ABB RAPID module: Operations.mod

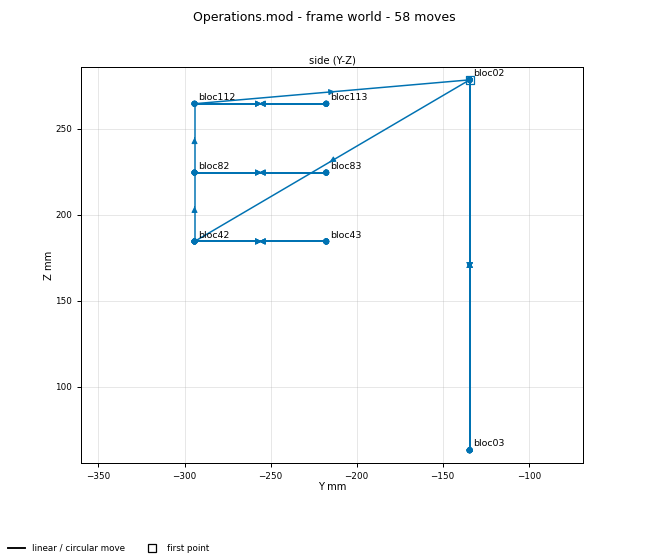
[picture p0: tool path of Operations.mod in frame world, 58 of 59 moves have a stored position in this frame; points joined in program order, loops and branches not executed]
MODULE Operations
 PROC GoHome()
  !
  VAR speeddata HomeSpeed:=[800,100,5000,1000];
  CONST jointtarget PlaceBloc0:=[[-88.65,-2.92,16.23,0,76.69,-88.65],[0,9E9,9E9,9E9,9E9,9E9]];
  MoveAbsJ PlaceBloc0,HomeSpeed,z1,EGP_40_N_N_B;
 ENDPROC
 PROC BuildWall()
  !
  VAR zonedata TransportZone:=[FALSE,5,7.5,7.5,0.75,7.5,0.75];
  VAR speeddata TransportSpeed:=[800,100,5000,1000];
  VAR speeddata PickSpeed:=[60,100,5000,1000];
  CONST robtarget bloc00:=[[-6.5,-340,128.58],[-0.183,-0.683,0.683,0.183],[-1,-1,-2,0],[0,9E9,9E9,9E9,9E9,9E9]];
  CONST robtarget bloc01:=[[-56.5,-340,41.98],[-0.183,-0.683,0.683,0.183],[-1,-1,-2,0],[0,9E9,9E9,9E9,9E9,9E9]];
  CONST robtarget bloc02:=[[211.67,-134.33,278.3],[0.6088,0.7934,0,0],[0,-1,-2,0],[0,9E9,9E9,9E9,9E9,9E9]];
  CONST robtarget bloc03:=[[211.67,-134.33,63.11],[0.6088,0.7934,0,0],[0,-1,-1,0],[0,9E9,9E9,9E9,9E9,9E9]];
  CONST robtarget bloc04:=[[506.47,-134.33,63.11],[0.6088,0.7934,0,0],[0,-1,-2,0],[0,9E9,9E9,9E9,9E9,9E9]];
  CONST robtarget bloc05:=[[506.47,-230.92,37.23],[0.6088,0.7934,0,0],[0,-1,-2,0],[0,9E9,9E9,9E9,9E9,9E9]];
  CONST robtarget bloc10:=[[-6.5,-340,128.58],[-0.183,-0.683,0.683,0.183],[-1,-1,-2,0],[0,9E9,9E9,9E9,9E9,9E9]];
  CONST robtarget bloc11:=[[-56.5,-340,41.98],[-0.183,-0.683,0.683,0.183],[-1,-1,-2,0],[0,9E9,9E9,9E9,9E9,9E9]];
  CONST robtarget bloc12:=[[211.67,-134.33,278.3],[0.6088,0.7934,0,0],[0,-1,-2,0],[0,9E9,9E9,9E9,9E9,9E9]];
  CONST robtarget bloc13:=[[211.67,-134.33,63.11],[0.6088,0.7934,0,0],[0,-1,-1,0],[0,9E9,9E9,9E9,9E9,9E9]];
  CONST robtarget bloc14:=[[424.47,-134.33,63.11],[0.6088,0.7934,0,0],[0,-1,-2,0],[0,9E9,9E9,9E9,9E9,9E9]];
  CONST robtarget bloc15:=[[424.47,-230.92,37.23],[0.6088,0.7934,0,0],[0,-1,-2,0],[0,9E9,9E9,9E9,9E9,9E9]];
  CONST robtarget bloc20:=[[-6.5,-340,128.58],[-0.183,-0.683,0.683,0.183],[-1,-1,-2,0],[0,9E9,9E9,9E9,9E9,9E9]];
  CONST robtarget bloc21:=[[-56.5,-340,41.98],[-0.183,-0.683,0.683,0.183],[-1,-1,-2,0],[0,9E9,9E9,9E9,9E9,9E9]];
  CONST robtarget bloc22:=[[211.67,-134.33,278.3],[0.6088,0.7934,0,0],[0,-1,-2,0],[0,9E9,9E9,9E9,9E9,9E9]];
  CONST robtarget bloc23:=[[211.67,-134.33,63.11],[0.6088,0.7934,0,0],[0,-1,-1,0],[0,9E9,9E9,9E9,9E9,9E9]];
  CONST robtarget bloc24:=[[342.47,-134.33,63.11],[0.6088,0.7934,0,0],[0,-1,-2,0],[0,9E9,9E9,9E9,9E9,9E9]];
  CONST robtarget bloc25:=[[342.47,-230.92,37.23],[0.6088,0.7934,0,0],[0,-1,-2,0],[0,9E9,9E9,9E9,9E9,9E9]];
  CONST robtarget bloc30:=[[-6.5,-340,128.58],[-0.183,-0.683,0.683,0.183],[-1,-1,-2,0],[0,9E9,9E9,9E9,9E9,9E9]];
  CONST robtarget bloc31:=[[-56.5,-340,41.98],[-0.183,-0.683,0.683,0.183],[-1,-1,-2,0],[0,9E9,9E9,9E9,9E9,9E9]];
  CONST robtarget bloc32:=[[211.67,-134.33,278.3],[0.6088,0.7934,0,0],[0,-1,-2,0],[0,9E9,9E9,9E9,9E9,9E9]];
  CONST robtarget bloc33:=[[211.67,-134.33,63.11],[0.6088,0.7934,0,0],[0,-1,-1,0],[0,9E9,9E9,9E9,9E9,9E9]];
  CONST robtarget bloc34:=[[260.47,-134.33,63.11],[0.6088,0.7934,0,0],[0,-1,-1,0],[0,9E9,9E9,9E9,9E9,9E9]];
  CONST robtarget bloc35:=[[260.47,-230.92,37.23],[0.6088,0.7934,0,0],[0,-2,-1,0],[0,9E9,9E9,9E9,9E9,9E9]];
  CONST robtarget bloc40:=[[5.76,-340,111.58],[-0.2706,-0.6533,0.6533,0.2706],[-1,-1,-2,0],[0,9E9,9E9,9E9,9E9,9E9]];
  CONST robtarget bloc41:=[[-64.95,-340,40.87],[-0.2706,-0.6533,0.6533,0.2706],[-1,-1,-2,0],[0,9E9,9E9,9E9,9E9,9E9]];
  CONST robtarget bloc42:=[[211.67,-294.18,184.42],[0,-0.7071,0.7071,0],[-1,0,-2,0],[0,9E9,9E9,9E9,9E9,9E9]];
  CONST robtarget bloc43:=[[211.67,-217.68,184.42],[0,-0.7071,0.7071,0],[-1,0,-2,0],[0,9E9,9E9,9E9,9E9,9E9]];
  CONST robtarget bloc44:=[[506.47,-217.68,184.42],[0,-0.7071,0.7071,0],[-1,0,-2,0],[0,9E9,9E9,9E9,9E9,9E9]];
  CONST robtarget bloc45:=[[506.47,-217.68,84.42],[0,-0.7071,0.7071,0],[-1,0,-2,0],[0,9E9,9E9,9E9,9E9,9E9]];
  CONST robtarget bloc50:=[[5.76,-340,111.58],[-0.2706,-0.6533,0.6533,0.2706],[-1,-1,-2,0],[0,9E9,9E9,9E9,9E9,9E9]];
  CONST robtarget bloc51:=[[-64.95,-340,40.87],[-0.2706,-0.6533,0.6533,0.2706],[-1,-1,-2,0],[0,9E9,9E9,9E9,9E9,9E9]];
  CONST robtarget bloc52:=[[211.67,-294.18,184.42],[0,-0.7071,0.7071,0],[-1,0,-2,0],[0,9E9,9E9,9E9,9E9,9E9]];
  CONST robtarget bloc53:=[[211.67,-217.68,184.42],[0,-0.7071,0.7071,0],[-1,0,-2,0],[0,9E9,9E9,9E9,9E9,9E9]];
  CONST robtarget bloc54:=[[424.47,-217.68,184.42],[0,-0.7071,0.7071,0],[-1,0,-2,0],[0,9E9,9E9,9E9,9E9,9E9]];
  CONST robtarget bloc55:=[[424.47,-217.68,84.42],[0,-0.7071,0.7071,0],[-1,0,-2,0],[0,9E9,9E9,9E9,9E9,9E9]];
  CONST robtarget bloc60:=[[5.76,-340,111.58],[-0.2706,-0.6533,0.6533,0.2706],[-1,-1,-2,0],[0,9E9,9E9,9E9,9E9,9E9]];
  CONST robtarget bloc61:=[[-64.95,-340,40.87],[-0.2706,-0.6533,0.6533,0.2706],[-1,-1,-2,0],[0,9E9,9E9,9E9,9E9,9E9]];
  CONST robtarget bloc62:=[[211.67,-294.18,184.42],[0,-0.7071,0.7071,0],[-1,0,-2,0],[0,9E9,9E9,9E9,9E9,9E9]];
  CONST robtarget bloc63:=[[211.67,-217.68,184.42],[0,-0.7071,0.7071,0],[-1,0,-2,0],[0,9E9,9E9,9E9,9E9,9E9]];
  CONST robtarget bloc64:=[[342.47,-217.68,184.42],[0,-0.7071,0.7071,0],[-1,0,-2,0],[0,9E9,9E9,9E9,9E9,9E9]];
  CONST robtarget bloc65:=[[342.47,-217.68,84.42],[0,-0.7071,0.7071,0],[-1,0,-2,0],[0,9E9,9E9,9E9,9E9,9E9]];
  CONST robtarget bloc70:=[[5.76,-340,111.58],[-0.2706,-0.6533,0.6533,0.2706],[-1,-1,-2,0],[0,9E9,9E9,9E9,9E9,9E9]];
  CONST robtarget bloc71:=[[-64.95,-340,40.87],[-0.2706,-0.6533,0.6533,0.2706],[-1,-1,-2,0],[0,9E9,9E9,9E9,9E9,9E9]];
  CONST robtarget bloc72:=[[211.67,-294.18,184.42],[0,-0.7071,0.7071,0],[-1,0,-2,0],[0,9E9,9E9,9E9,9E9,9E9]];
  CONST robtarget bloc73:=[[211.67,-217.68,184.42],[0,-0.7071,0.7071,0],[-1,0,-2,0],[0,9E9,9E9,9E9,9E9,9E9]];
  CONST robtarget bloc74:=[[260.47,-217.68,184.42],[0,-0.7071,0.7071,0],[-1,0,-2,0],[0,9E9,9E9,9E9,9E9,9E9]];
  CONST robtarget bloc75:=[[260.47,-217.68,84.42],[0,-0.7071,0.7071,0],[-1,0,-2,0],[0,9E9,9E9,9E9,9E9,9E9]];
  CONST robtarget bloc80:=[[5.76,-340,111.58],[-0.2706,-0.6533,0.6533,0.2706],[-1,-1,-2,0],[0,9E9,9E9,9E9,9E9,9E9]];
  CONST robtarget bloc81:=[[-64.95,-340,40.87],[-0.2706,-0.6533,0.6533,0.2706],[-1,-1,-2,0],[0,9E9,9E9,9E9,9E9,9E9]];
  CONST robtarget bloc82:=[[211.67,-294.18,224.42],[0,-0.7071,0.7071,0],[-1,0,-2,0],[0,9E9,9E9,9E9,9E9,9E9]];
  CONST robtarget bloc83:=[[211.67,-217.68,224.42],[0,-0.7071,0.7071,0],[-1,0,-2,0],[0,9E9,9E9,9E9,9E9,9E9]];
  CONST robtarget bloc84:=[[466.47,-217.68,224.42],[0,-0.7071,0.7071,0],[-1,0,-2,0],[0,9E9,9E9,9E9,9E9,9E9]];
  CONST robtarget bloc85:=[[466.47,-217.68,124.42],[0,-0.7071,0.7071,0],[-1,0,-2,0],[0,9E9,9E9,9E9,9E9,9E9]];
  CONST robtarget bloc90:=[[5.76,-340,111.58],[-0.2706,-0.6533,0.6533,0.2706],[-1,-1,-2,0],[0,9E9,9E9,9E9,9E9,9E9]];
  CONST robtarget bloc91:=[[-64.95,-340,40.87],[-0.2706,-0.6533,0.6533,0.2706],[-1,-1,-2,0],[0,9E9,9E9,9E9,9E9,9E9]];
  CONST robtarget bloc92:=[[211.67,-294.18,224.42],[0,-0.7071,0.7071,0],[-1,0,-2,0],[0,9E9,9E9,9E9,9E9,9E9]];
  CONST robtarget bloc93:=[[211.67,-217.68,224.42],[0,-0.7071,0.7071,0],[-1,0,-2,0],[0,9E9,9E9,9E9,9E9,9E9]];
  CONST robtarget bloc94:=[[384.47,-217.68,224.42],[0,-0.7071,0.7071,0],[-1,0,-2,0],[0,9E9,9E9,9E9,9E9,9E9]];
  CONST robtarget bloc95:=[[384.47,-217.68,124.42],[0,-0.7071,0.7071,0],[-1,0,-2,0],[0,9E9,9E9,9E9,9E9,9E9]];
  CONST robtarget bloc100:=[[5.76,-340,111.58],[-0.2706,-0.6533,0.6533,0.2706],[-1,-1,-2,0],[0,9E9,9E9,9E9,9E9,9E9]];
  CONST robtarget bloc101:=[[-64.95,-340,40.87],[-0.2706,-0.6533,0.6533,0.2706],[-1,-1,-2,0],[0,9E9,9E9,9E9,9E9,9E9]];
  CONST robtarget bloc102:=[[211.67,-294.18,224.42],[0,-0.7071,0.7071,0],[-1,0,-2,0],[0,9E9,9E9,9E9,9E9,9E9]];
  CONST robtarget bloc103:=[[211.67,-217.68,224.42],[0,-0.7071,0.7071,0],[-1,0,-2,0],[0,9E9,9E9,9E9,9E9,9E9]];
  CONST robtarget bloc104:=[[302.47,-217.68,224.42],[0,-0.7071,0.7071,0],[-1,0,-2,0],[0,9E9,9E9,9E9,9E9,9E9]];
  CONST robtarget bloc105:=[[302.47,-217.68,124.42],[0,-0.7071,0.7071,0],[-1,0,-2,0],[0,9E9,9E9,9E9,9E9,9E9]];
  CONST robtarget bloc110:=[[5.76,-340,111.58],[-0.2706,-0.6533,0.6533,0.2706],[-1,-1,-2,0],[0,9E9,9E9,9E9,9E9,9E9]];
  CONST robtarget bloc111:=[[-64.95,-340,40.87],[-0.2706,-0.6533,0.6533,0.2706],[-1,-1,-2,0],[0,9E9,9E9,9E9,9E9,9E9]];
  CONST robtarget bloc112:=[[211.67,-294.18,264.42],[0,-0.7071,0.7071,0],[-1,0,-2,0],[0,9E9,9E9,9E9,9E9,9E9]];
  CONST robtarget bloc113:=[[211.67,-217.68,264.42],[0,-0.7071,0.7071,0],[-1,0,-2,0],[0,9E9,9E9,9E9,9E9,9E9]];
  CONST robtarget bloc114:=[[426.47,-217.68,264.42],[0,-0.7071,0.7071,0],[-1,0,-2,0],[0,9E9,9E9,9E9,9E9,9E9]];
  CONST robtarget bloc115:=[[426.47,-217.68,164.42],[0,-0.7071,0.7071,0],[-1,0,-2,0],[0,9E9,9E9,9E9,9E9,9E9]];
  CONST robtarget bloc120:=[[5.76,-340,111.58],[-0.2706,-0.6533,0.6533,0.2706],[-1,-1,-2,0],[0,9E9,9E9,9E9,9E9,9E9]];
  CONST robtarget bloc121:=[[-64.95,-340,40.87],[-0.2706,-0.6533,0.6533,0.2706],[-1,-1,-2,0],[0,9E9,9E9,9E9,9E9,9E9]];
  CONST robtarget bloc122:=[[211.67,-294.18,264.42],[0,-0.7071,0.7071,0],[-1,0,-2,0],[0,9E9,9E9,9E9,9E9,9E9]];
  CONST robtarget bloc123:=[[211.67,-217.68,264.42],[0,-0.7071,0.7071,0],[-1,0,-2,0],[0,9E9,9E9,9E9,9E9,9E9]];
  CONST robtarget bloc124:=[[344.47,-217.68,264.42],[0,-0.7071,0.7071,0],[-1,0,-2,0],[0,9E9,9E9,9E9,9E9,9E9]];
  CONST robtarget bloc125:=[[344.47,-217.68,164.42],[0,-0.7071,0.7071,0],[-1,0,-2,0],[0,9E9,9E9,9E9,9E9,9E9]];
  CONST robtarget bloc130:=[[5.76,-340,111.58],[-0.2706,-0.6533,0.6533,0.2706],[-1,-1,-2,0],[0,9E9,9E9,9E9,9E9,9E9]];
  CONST robtarget bloc131:=[[-64.95,-340,40.87],[-0.2706,-0.6533,0.6533,0.2706],[-1,-1,-2,0],[0,9E9,9E9,9E9,9E9,9E9]];
  CONST robtarget bloc132:=[[211.67,-294.18,264.42],[0,-0.7071,0.7071,0],[-1,0,-2,0],[0,9E9,9E9,9E9,9E9,9E9]];
  CONST robtarget bloc133:=[[211.67,-217.68,264.42],[0,-0.7071,0.7071,0],[-1,0,-2,0],[0,9E9,9E9,9E9,9E9,9E9]];
  CONST robtarget bloc134:=[[262.47,-217.68,264.42],[0,-0.7071,0.7071,0],[-1,0,-2,0],[0,9E9,9E9,9E9,9E9,9E9]];
  CONST robtarget bloc135:=[[262.47,-217.68,164.42],[0,-0.7071,0.7071,0],[-1,0,-2,0],[0,9E9,9E9,9E9,9E9,9E9]];
  StartGripper;
  PathAccLim TRUE \AccMax:=0.6, TRUE \DecelMax:=0.6;
  TakeBloc bloc00, bloc01, EGP_40_N_N_B, TransportSpeed, PickSpeed;
  MoveL bloc02,TransportSpeed,TransportZone,EGP_40_N_N_B\WObj:=WObj0;
  MoveL bloc03,TransportSpeed,TransportZone,EGP_40_N_N_B\WObj:=WObj0;
  ReleaseBloc bloc04, bloc05, EGP_40_N_N_B, TransportSpeed, PickSpeed;
  MoveL bloc03,TransportSpeed,TransportZone,EGP_40_N_N_B\WObj:=WObj0;
  MoveL bloc02,TransportSpeed,TransportZone,EGP_40_N_N_B\WObj:=WObj0;
  TakeBloc bloc10, bloc11, EGP_40_N_N_B, TransportSpeed, PickSpeed;
  MoveL bloc12,TransportSpeed,TransportZone,EGP_40_N_N_B\WObj:=WObj0;
  MoveL bloc13,TransportSpeed,TransportZone,EGP_40_N_N_B\WObj:=WObj0;
  ReleaseBloc bloc14, bloc15, EGP_40_N_N_B, TransportSpeed, PickSpeed;
  MoveL bloc13,TransportSpeed,TransportZone,EGP_40_N_N_B\WObj:=WObj0;
  MoveL bloc12,TransportSpeed,TransportZone,EGP_40_N_N_B\WObj:=WObj0;
  TakeBloc bloc20, bloc21, EGP_40_N_N_B, TransportSpeed, PickSpeed;
  MoveL bloc22,TransportSpeed,TransportZone,EGP_40_N_N_B\WObj:=WObj0;
  MoveL bloc23,TransportSpeed,TransportZone,EGP_40_N_N_B\WObj:=WObj0;
  ReleaseBloc bloc24, bloc25, EGP_40_N_N_B, TransportSpeed, PickSpeed;
  MoveL bloc23,TransportSpeed,TransportZone,EGP_40_N_N_B\WObj:=WObj0;
  MoveL bloc22,TransportSpeed,TransportZone,EGP_40_N_N_B\WObj:=WObj0;
  TakeBloc bloc30, bloc31, EGP_40_N_N_B, TransportSpeed, PickSpeed;
  MoveL bloc32,TransportSpeed,TransportZone,EGP_40_N_N_B\WObj:=WObj0;
  MoveL bloc33,TransportSpeed,TransportZone,EGP_40_N_N_B\WObj:=WObj0;
  ReleaseBloc bloc34, bloc35, EGP_40_N_N_B, TransportSpeed, PickSpeed;
  MoveL bloc33,TransportSpeed,TransportZone,EGP_40_N_N_B\WObj:=WObj0;
  MoveL bloc32,TransportSpeed,TransportZone,EGP_40_N_N_B\WObj:=WObj0;
  TakeBloc bloc40, bloc41, EGP_40_N_N_B, TransportSpeed, PickSpeed;
  MoveL bloc42,TransportSpeed,TransportZone,EGP_40_N_N_B\WObj:=WObj0;
  MoveL bloc43,TransportSpeed,TransportZone,EGP_40_N_N_B\WObj:=WObj0;
  ReleaseBloc bloc44, bloc45, EGP_40_N_N_B, TransportSpeed, PickSpeed;
  MoveL bloc43,TransportSpeed,TransportZone,EGP_40_N_N_B\WObj:=WObj0;
  MoveL bloc42,TransportSpeed,TransportZone,EGP_40_N_N_B\WObj:=WObj0;
  TakeBloc bloc50, bloc51, EGP_40_N_N_B, TransportSpeed, PickSpeed;
  MoveL bloc52,TransportSpeed,TransportZone,EGP_40_N_N_B\WObj:=WObj0;
  MoveL bloc53,TransportSpeed,TransportZone,EGP_40_N_N_B\WObj:=WObj0;
  ReleaseBloc bloc54, bloc55, EGP_40_N_N_B, TransportSpeed, PickSpeed;
  MoveL bloc53,TransportSpeed,TransportZone,EGP_40_N_N_B\WObj:=WObj0;
  MoveL bloc52,TransportSpeed,TransportZone,EGP_40_N_N_B\WObj:=WObj0;
  TakeBloc bloc60, bloc61, EGP_40_N_N_B, TransportSpeed, PickSpeed;
  MoveL bloc62,TransportSpeed,TransportZone,EGP_40_N_N_B\WObj:=WObj0;
  MoveL bloc63,TransportSpeed,TransportZone,EGP_40_N_N_B\WObj:=WObj0;
  ReleaseBloc bloc64, bloc65, EGP_40_N_N_B, TransportSpeed, PickSpeed;
  MoveL bloc63,TransportSpeed,TransportZone,EGP_40_N_N_B\WObj:=WObj0;
  MoveL bloc62,TransportSpeed,TransportZone,EGP_40_N_N_B\WObj:=WObj0;
  TakeBloc bloc70, bloc71, EGP_40_N_N_B, TransportSpeed, PickSpeed;
  MoveL bloc72,TransportSpeed,TransportZone,EGP_40_N_N_B\WObj:=WObj0;
  MoveL bloc73,TransportSpeed,TransportZone,EGP_40_N_N_B\WObj:=WObj0;
  ReleaseBloc bloc74, bloc75, EGP_40_N_N_B, TransportSpeed, PickSpeed;
  MoveL bloc73,TransportSpeed,TransportZone,EGP_40_N_N_B\WObj:=WObj0;
  MoveL bloc72,TransportSpeed,TransportZone,EGP_40_N_N_B\WObj:=WObj0;
  TakeBloc bloc80, bloc81, EGP_40_N_N_B, TransportSpeed, PickSpeed;
  MoveL bloc82,TransportSpeed,TransportZone,EGP_40_N_N_B\WObj:=WObj0;
  MoveL bloc83,TransportSpeed,TransportZone,EGP_40_N_N_B\WObj:=WObj0;
  ReleaseBloc bloc84, bloc85, EGP_40_N_N_B, TransportSpeed, PickSpeed;
  MoveL bloc83,TransportSpeed,TransportZone,EGP_40_N_N_B\WObj:=WObj0;
  MoveL bloc82,TransportSpeed,TransportZone,EGP_40_N_N_B\WObj:=WObj0;
  TakeBloc bloc90, bloc91, EGP_40_N_N_B, TransportSpeed, PickSpeed;
  MoveL bloc92,TransportSpeed,TransportZone,EGP_40_N_N_B\WObj:=WObj0;
  MoveL bloc93,TransportSpeed,TransportZone,EGP_40_N_N_B\WObj:=WObj0;
  ReleaseBloc bloc94, bloc95, EGP_40_N_N_B, TransportSpeed, PickSpeed;
  MoveL bloc93,TransportSpeed,TransportZone,EGP_40_N_N_B\WObj:=WObj0;
  MoveL bloc92,TransportSpeed,TransportZone,EGP_40_N_N_B\WObj:=WObj0;
  TakeBloc bloc100, bloc101, EGP_40_N_N_B, TransportSpeed, PickSpeed;
  MoveL bloc102,TransportSpeed,TransportZone,EGP_40_N_N_B\WObj:=WObj0;
  MoveL bloc103,TransportSpeed,TransportZone,EGP_40_N_N_B\WObj:=WObj0;
  ReleaseBloc bloc104, bloc105, EGP_40_N_N_B, TransportSpeed, PickSpeed;
  MoveL bloc103,TransportSpeed,TransportZone,EGP_40_N_N_B\WObj:=WObj0;
  MoveL bloc102,TransportSpeed,TransportZone,EGP_40_N_N_B\WObj:=WObj0;
  TakeBloc bloc110, bloc111, EGP_40_N_N_B, TransportSpeed, PickSpeed;
  MoveL bloc112,TransportSpeed,TransportZone,EGP_40_N_N_B\WObj:=WObj0;
  MoveL bloc113,TransportSpeed,TransportZone,EGP_40_N_N_B\WObj:=WObj0;
  ReleaseBloc bloc114, bloc115, EGP_40_N_N_B, TransportSpeed, PickSpeed;
  MoveL bloc113,TransportSpeed,TransportZone,EGP_40_N_N_B\WObj:=WObj0;
  MoveL bloc112,TransportSpeed,TransportZone,EGP_40_N_N_B\WObj:=WObj0;
  TakeBloc bloc120, bloc121, EGP_40_N_N_B, TransportSpeed, PickSpeed;
  MoveL bloc122,TransportSpeed,TransportZone,EGP_40_N_N_B\WObj:=WObj0;
  MoveL bloc123,TransportSpeed,TransportZone,EGP_40_N_N_B\WObj:=WObj0;
  ReleaseBloc bloc124, bloc125, EGP_40_N_N_B, TransportSpeed, PickSpeed;
  MoveL bloc123,TransportSpeed,TransportZone,EGP_40_N_N_B\WObj:=WObj0;
  MoveL bloc122,TransportSpeed,TransportZone,EGP_40_N_N_B\WObj:=WObj0;
  TakeBloc bloc130, bloc131, EGP_40_N_N_B, TransportSpeed, PickSpeed;
  MoveL bloc132,TransportSpeed,TransportZone,EGP_40_N_N_B\WObj:=WObj0;
  MoveL bloc133,TransportSpeed,TransportZone,EGP_40_N_N_B\WObj:=WObj0;
  ReleaseBloc bloc134, bloc135, EGP_40_N_N_B, TransportSpeed, PickSpeed;
  MoveL bloc133,TransportSpeed,TransportZone,EGP_40_N_N_B\WObj:=WObj0;
  MoveL bloc132,TransportSpeed,TransportZone,EGP_40_N_N_B\WObj:=WObj0;
  MoveL bloc22,TransportSpeed,TransportZone,EGP_40_N_N_B\WObj:=WObj0;
  MoveL bloc23,TransportSpeed,TransportZone,EGP_40_N_N_B\WObj:=WObj0;
  TakeBloc bloc24, bloc25, EGP_40_N_N_B, TransportSpeed, PickSpeed;
  ShutdownGripper;
 ENDPROC
ENDMODULE
